# EPICS substitutions: db/core/ecmcEcSlave.substitutions
file "ecmcEcSlave.template"
{
    pattern {}
            {}
}
